// TIA Portal V18 export
DATA_BLOCK "ActualHWAlarmsList"   // DB10001
{ S7_Optimized_Access := 'FALSE' }
VERSION : 0.1
// stored: AutoNumber false, DBAccessibleFromOPCUA true, IsOnlyStoredInLoadMemory false, IsWriteProtectedInAS false
   VAR
      iActiveFaults : DInt;
      iWriteIndex : Int;
      Log { S7_SetPoint := 'True'} : Array[0..99] of "UDT_HWAlarmEntry";
   END_VAR
BEGIN
END_DATA_BLOCK
